// TIA Portal V19 export
// export: Created 2024-12-12T07:14:08.2418782Z, ExportSetting WithDefaults, DisplayName Totally Integrated Automation Portal, DisplayVersion V19 Update 1, DisplayName TIA Portal Openness, DisplayVersion V19 Update 1, DisplayName TIA Portal Version Control Interface, DisplayVersion V19, DisplayName SINAMICS Startdrive Advanced, DisplayVersion V19, DisplayName SINAMICS DCC, DisplayVersion V19, DisplayName SINAMICS Startdrive G130, G150, S120, S150, SINAMICS MV, G220, S200, S210, DisplayVersion V19, DisplayName SINAMICS Startdrive G110M, G120, G120C, G120D, G120P, G115D, DisplayVersion V19, DisplayName STEP 7 Professional, DisplayVersion V19 Update 1, DisplayName STEP 7 Safety, DisplayVersion V19 Update 1, DisplayName WinCC Advanced, DisplayVersion V19 Update 1, DisplayName WinCC Advanced / Unified PC, DisplayVersion V19 Update 1
DATA_BLOCK "DP1"   // DB30
{ S7_Optimized_Access := 'TRUE' }
VERSION : 0.1
// stored: AutoNumber true, DBAccessibleFromOPCUA true, DBAccessibleFromWebserver true, InstanceOfName DP_Exchange, InstanceOfType UDT, IsOnlyStoredInLoadMemory false, IsWriteProtectedInAS false
"DP_Exchange"
   // VAR RETAIN
   //    ExchangeToChain : "DP_Exchange_ToChain";
   //    ExchangeFromChain : "DP_Exchange_FromChain";
   //    Std : "DP_Exchange_Std";
   // END_VAR
BEGIN
   ExchangeToChain.Communication.RunMode := TRUE;
   ExchangeToChain.Communication.ConnectionFaulted := FALSE;
   ExchangeToChain.Work.Depositor := FALSE;
   ExchangeToChain.Work.TempDetect := FALSE;
   ExchangeToChain.Work.Vibrators := FALSE;
   ExchangeToChain.WorkedBy.Depositor := FALSE;
   ExchangeToChain.WorkedBy.TempDetect := FALSE;
   ExchangeToChain.WorkedBy.Vibrators := FALSE;
   ExchangeToChain.OutChainObstruction.Depositor := TRUE;
   ExchangeToChain.OutChainObstruction.TempDetect := TRUE;
   ExchangeToChain.OutChainObstruction.Vibrators := TRUE;
   ExchangeToChain.TimeWork.Depositor := 0;
   ExchangeToChain.TimeWork.Vibrator1 := 0;
   ExchangeToChain.TimeWork.Vibrator2 := 0;
   ExchangeToChain.TimeWork.VIbrator3 := 0;
   ExchangeToChain.AlmOKImmStopChain := TRUE;
   ExchangeToChain.Set_StrobeWorkReq := FALSE;
   ExchangeToChain.Set_StrobeWorkReqMouldBlock := FALSE;
   ExchangeToChain.RejByCycleInterruption := FALSE;
   ExchangeToChain.ChangeSpeedEna := TRUE;
   ExchangeToChain.MarkedByOpe := FALSE;
   ExchangeToChain.PresMould := FALSE;
   ExchangeToChain.Starved := FALSE;
   ExchangeToChain.DepositorEnabled := TRUE;
   ExchangeToChain.TempDetectorEnabled := TRUE;
   ExchangeToChain.LocalModeReq := FALSE;
   ExchangeToChain.Weight_StopInPhaseReq := TRUE;
   ExchangeToChain.Weight_AcusticReq := TRUE;
   ExchangeToChain.NoDoseAllowed := FALSE;
   ExchangeToChain."Dint"[0..4] := 0;
   ExchangeToChain.TempDetect_ScaledValue := 25.82104;
   ExchangeToChain.VMasterAtCycleEnd := 312.455;
   ExchangeToChain.VMasterRegPos := 0.0;
   ExchangeToChain.Infeed_VMasterRegPos1 := 0.0;
   ExchangeToChain.Infeed_VMasterRegPos2 := 0.0;
   ExchangeToChain.Outfeed_VMasterRegPos1 := 0.0;
   ExchangeToChain.Outfeed_VMasterRegPos2 := 0.0;
   ExchangeFromChain.Communication.RunMode := TRUE;
   ExchangeFromChain.Communication.ConnectionFaulted := FALSE;
   ExchangeFromChain.Chain.EnableMove := TRUE;
   ExchangeFromChain.Chain.StrobeWorkReq := FALSE;
   ExchangeFromChain.Chain.StrobeWorkReqMouldBlock := FALSE;
   ExchangeFromChain.Chain.CheckObstruction := FALSE;
   ExchangeFromChain.Chain.MoveInMan := FALSE;
   ExchangeFromChain.Chain.VMasterInPosition := TRUE;
   ExchangeFromChain.Chain.VMasterAtSpeed := FALSE;
   ExchangeFromChain.Chain.Cfg_1Jog_0Move := FALSE;
   ExchangeFromChain.ReqWork.Depositor := FALSE;
   ExchangeFromChain.ReqWork.TempDetect := FALSE;
   ExchangeFromChain.ReqWork.Vibrators := TRUE;
   ExchangeFromChain.SetWorkedBy.Depositor := FALSE;
   ExchangeFromChain.SetWorkedBy.TempDetect := FALSE;
   ExchangeFromChain.SetWorkedBy.Vibrators := FALSE;
   ExchangeFromChain.Set_MarkedByOpe := FALSE;
   ExchangeFromChain.Set_RejByCycleInterruption := FALSE;
   ExchangeFromChain.ChangeSpeedReq := FALSE;
   ExchangeFromChain.LocalModeActived := FALSE;
   ExchangeFromChain.LocalAbortReq := FALSE;
   ExchangeFromChain.Selected := TRUE;
   ExchangeFromChain."Dint"[0..4] := 0;
   ExchangeFromChain.SetPointSpeed := 25.0;
   ExchangeFromChain.ActualSpeed := 0.0;
   Std.ExchangeToGlobal.Communication.RunMode := TRUE;
   Std.ExchangeToGlobal.Communication.ConnectionFaulted := FALSE;
   Std.ExchangeToGlobal.Gen.Communication := FALSE;
   Std.ExchangeToGlobal.Gen.Selected := TRUE;
   Std.ExchangeToGlobal.Gen.Extracted := FALSE;
   Std.ExchangeToGlobal.Gen.EnaReq := FALSE;
   Std.ExchangeToGlobal.Gen.StaReq := FALSE;
   Std.ExchangeToGlobal.Gen.Started := FALSE;
   Std.ExchangeToGlobal.Gen.Unsuspended := FALSE;
   Std.ExchangeToGlobal.Gen.Ena_Suspended := TRUE;
   Std.ExchangeToGlobal.Gen.sts_Starting := FALSE;
   Std.ExchangeToGlobal.Gen.sts_Stopping := FALSE;
   Std.ExchangeToGlobal.Gen.sts_Aborting := FALSE;
   Std.ExchangeToGlobal.Gen.sts_Suspending := FALSE;
   Std.ExchangeToGlobal.Gen.sts_Unsuspending := FALSE;
   Std.ExchangeToGlobal.Gen.sts_Execute := FALSE;
   Std.ExchangeToGlobal.Gen.sts_Idle := TRUE;
   Std.ExchangeToGlobal.Gen.sts_Stopped := FALSE;
   Std.ExchangeToGlobal.Gen.sts_Aborted := FALSE;
   Std.ExchangeToGlobal.Gen.sts_Suspended := FALSE;
   Std.ExchangeToGlobal.Gen.sts_ModeManual := FALSE;
   Std.ExchangeToGlobal.Gen.sts_ModeAutomatic := TRUE;
   Std.ExchangeToGlobal.Gen.NewAlm := FALSE;
   Std.ExchangeToGlobal.Gen.NewSign := FALSE;
   Std.ExchangeToGlobal.Gen.RecipeOnlineLoadDone := FALSE;
   Std.ExchangeToGlobal.Gen.RecipeOnlineSaveDone := FALSE;
   Std.ExchangeToGlobal.Gen.RecipeOfflineLoadDone := FALSE;
   Std.ExchangeToGlobal.Gen.RecipeOfflineSaveDone := FALSE;
   Std.ExchangeToGlobal.Gen.LastHmiDataLoadDone := FALSE;
   Std.ExchangeToGlobal.Gen.LastHmiDataSaveDone := FALSE;
   Std.ExchangeToGlobal.Gen.InverterDiagnosticDone := FALSE;
   Std.ExchangeToGlobal.Gen.CmdMode := 1;
   Std.ExchangeToGlobal.Gen.Mode := 1;
   Std.ExchangeToGlobal.Gen.DisableEnaPbt := 0;
   Std.ExchangeToGlobal.Input.StaPbt := FALSE;
   Std.ExchangeToGlobal.Input.StoPbt := FALSE;
   Std.ExchangeToGlobal.Input.RstPbt := FALSE;
   Std.ExchangeToGlobal.Input.EnaPbt := FALSE;
   Std.ExchangeToGlobal.Input._4 := FALSE;
   Std.ExchangeToGlobal.Input._5 := FALSE;
   Std.ExchangeToGlobal.Input._6 := FALSE;
   Std.ExchangeToGlobal.Input._7 := FALSE;
   Std.ExchangeToGlobal.Input._8 := FALSE;
   Std.ExchangeToGlobal.Input._9 := FALSE;
   Std.ExchangeToGlobal.Input._10 := FALSE;
   Std.ExchangeToGlobal.Input._11 := FALSE;
   Std.ExchangeToGlobal.Input._12 := FALSE;
   Std.ExchangeToGlobal.Input._13 := FALSE;
   Std.ExchangeToGlobal.Input._14 := FALSE;
   Std.ExchangeToGlobal.Input._15 := FALSE;
   Std.ExchangeToGlobal.AlmOk.ThSwitch := TRUE;
   Std.ExchangeToGlobal.AlmOk.SafeComm := TRUE;
   Std.ExchangeToGlobal.AlmOk.SafeEmg := TRUE;
   Std.ExchangeToGlobal.AlmOk.SafeGuards := TRUE;
   Std.ExchangeToGlobal.AlmOk.GtaAirGroup := TRUE;
   Std.ExchangeToGlobal.AlmOk.Major := TRUE;
   Std.ExchangeToGlobal.AlmOk.Minor := TRUE;
   Std.ExchangeToGlobal.AlmOk.Spare07 := TRUE;
   Std.ExchangeToGlobal.AlmOk.Spare08 := TRUE;
   Std.ExchangeToGlobal.AlmOk.Spare09 := TRUE;
   Std.ExchangeToGlobal.AlmOk.Spare10 := TRUE;
   Std.ExchangeToGlobal.AlmOk.Spare11 := TRUE;
   Std.ExchangeToGlobal.AlmOk.Spare12 := TRUE;
   Std.ExchangeToGlobal.AlmOk.Spare13 := TRUE;
   Std.ExchangeToGlobal.AlmOk.Spare14 := TRUE;
   Std.ExchangeToGlobal.AlmOk.Spare15 := TRUE;
   Std.ExchangeToGlobal.AlmOk.Spare16 := TRUE;
   Std.ExchangeToGlobal.AlmOk.Spare17 := TRUE;
   Std.ExchangeToGlobal.AlmOk.Spare18 := TRUE;
   Std.ExchangeToGlobal.AlmOk.Spare19 := TRUE;
   Std.ExchangeToGlobal.AlmOk.Spare20 := TRUE;
   Std.ExchangeToGlobal.AlmOk.Spare21 := TRUE;
   Std.ExchangeToGlobal.AlmOk.Spare22 := TRUE;
   Std.ExchangeToGlobal.AlmOk.Spare23 := TRUE;
   Std.ExchangeToGlobal.AlmOk.Spare24 := TRUE;
   Std.ExchangeToGlobal.AlmOk.Spare25 := TRUE;
   Std.ExchangeToGlobal.AlmOk.Spare26 := TRUE;
   Std.ExchangeToGlobal.AlmOk.Spare27 := TRUE;
   Std.ExchangeToGlobal.AlmOk.Spare28 := TRUE;
   Std.ExchangeToGlobal.AlmOk.Spare29 := TRUE;
   Std.ExchangeToGlobal.AlmOk.Spare30 := TRUE;
   Std.ExchangeToGlobal.AlmOk.Spare31 := TRUE;
   Std.ExchangeToGlobal.AlmCauseOk.Ope := TRUE;
   Std.ExchangeToGlobal.AlmCauseOk.Ust := TRUE;
   Std.ExchangeToGlobal.AlmCauseOk.Dst := TRUE;
   Std.ExchangeToGlobal.AlmCauseOk.Ext := TRUE;
   Std.ExchangeToGlobal.AlmCauseOk.Mac := TRUE;
   Std.ExchangeToGlobal.AlmCauseOk.Spare05 := TRUE;
   Std.ExchangeToGlobal.AlmCauseOk.Spare06 := TRUE;
   Std.ExchangeToGlobal.AlmCauseOk.Spare07 := TRUE;
   Std.ExchangeToGlobal.AlmCauseOk.Spare08 := TRUE;
   Std.ExchangeToGlobal.AlmCauseOk.Spare09 := TRUE;
   Std.ExchangeToGlobal.AlmCauseOk.Spare10 := TRUE;
   Std.ExchangeToGlobal.AlmCauseOk.Spare11 := TRUE;
   Std.ExchangeToGlobal.AlmCauseOk.Spare12 := TRUE;
   Std.ExchangeToGlobal.AlmCauseOk.Spare13 := TRUE;
   Std.ExchangeToGlobal.AlmCauseOk.Spare14 := TRUE;
   Std.ExchangeToGlobal.AlmCauseOk.Spare15 := TRUE;
   Std.ExchangeToGlobal.AlmCauseOk.Spare16 := TRUE;
   Std.ExchangeToGlobal.AlmCauseOk.Spare17 := TRUE;
   Std.ExchangeToGlobal.AlmCauseOk.Spare18 := TRUE;
   Std.ExchangeToGlobal.AlmCauseOk.Spare19 := TRUE;
   Std.ExchangeToGlobal.AlmCauseOk.Spare20 := TRUE;
   Std.ExchangeToGlobal.AlmCauseOk.Spare21 := TRUE;
   Std.ExchangeToGlobal.AlmCauseOk.Spare22 := TRUE;
   Std.ExchangeToGlobal.AlmCauseOk.Spare23 := TRUE;
   Std.ExchangeToGlobal.AlmCauseOk.Spare24 := TRUE;
   Std.ExchangeToGlobal.AlmCauseOk.Spare25 := TRUE;
   Std.ExchangeToGlobal.AlmCauseOk.Spare26 := TRUE;
   Std.ExchangeToGlobal.AlmCauseOk.Spare27 := TRUE;
   Std.ExchangeToGlobal.AlmCauseOk.Spare28 := TRUE;
   Std.ExchangeToGlobal.AlmCauseOk.Spare29 := TRUE;
   Std.ExchangeToGlobal.AlmCauseOk.Spare30 := TRUE;
   Std.ExchangeToGlobal.AlmCauseOk.Spare31 := TRUE;
   Std.ExchangeToGlobal.AlmBannerFbk.FirstAlmDetection := FALSE;
   Std.ExchangeToGlobal.AlmBannerFbk.AlmPriority := 100;
   Std.ExchangeToGlobal.AlmBannerFbk.AlmCategory := -1;
   Std.ExchangeToGlobal.AlmBannerFbk.AlmCause := -1;
   Std.ExchangeToGlobal.AlmBannerFbk.AlmID := -1;
   Std.ExchangeToGlobal.AlmBannerFbk.GlobalAbsTime := 0;
   Std.ExchangeToGlobal.SignBannerFbk.SignPriority := 100;
   Std.ExchangeToGlobal.SignBannerFbk.SignCategory := -1;
   Std.ExchangeToGlobal.SignBannerFbk.SignID := -1;
   Std.ExchangeToGlobal.ExtCPU.PushButton.StaPbt := FALSE;
   Std.ExchangeToGlobal.ExtCPU.PushButton.StoPbt := FALSE;
   Std.ExchangeToGlobal.ExtCPU.PushButton.RstPbt := FALSE;
   Std.ExchangeToGlobal.ExtCPU.PushButton.EnaPbt := FALSE;
   Std.ExchangeToGlobal.ExtCPU.PushButton.EnaReq := FALSE;
   Std.ExchangeToGlobal.ExtCPU.PushButton.EnaStaReq := FALSE;
   Std.ExchangeToGlobal.ExtCPU.DeviceDiagDone := TRUE;
   Std.ExchangeToGlobal.ExtCPU.InverterDiagDone := FALSE;
   Std.ExchangeToGlobal.LightSiren.Cfg_StaPbt := 12515;
   Std.ExchangeToGlobal.LightSiren.Cfg_RstPbt := -1;
   Std.ExchangeToGlobal.LightSiren.Cfg_EnaPbt := 12515;
   Std.ExchangeToGlobal.LightSiren.Cfg_Siren := 3;
   Std.ExchangeToGlobal.LightSiren.Cfg_Stack := 3;
   Std.ExchangeToGlobal.LightSiren.Steady.StaPbtLgh := FALSE;
   Std.ExchangeToGlobal.LightSiren.Steady.RstPbtLgh := FALSE;
   Std.ExchangeToGlobal.LightSiren.Steady.EnaPbtLgh := FALSE;
   Std.ExchangeToGlobal.LightSiren.Steady.Siren := FALSE;
   Std.ExchangeToGlobal.LightSiren.Steady.YelStkLgh := FALSE;
   Std.ExchangeToGlobal.LightSiren.Steady.BluStkLgh := FALSE;
   Std.ExchangeToGlobal.LightSiren.Steady.GrnStkLgh := FALSE;
   Std.ExchangeToGlobal.LightSiren.Steady.WhtStkLgh := FALSE;
   Std.ExchangeToGlobal.LightSiren.Steady.Cust1_StaPbtLgh := FALSE;
   Std.ExchangeToGlobal.LightSiren.Steady.Cust1_RstPbtLgh := FALSE;
   Std.ExchangeToGlobal.LightSiren.Steady.Cust1_Siren := FALSE;
   Std.ExchangeToGlobal.LightSiren.Steady.Cust1_RedStkLgh := FALSE;
   Std.ExchangeToGlobal.LightSiren.Steady.Cust1_OngStkLgh := FALSE;
   Std.ExchangeToGlobal.LightSiren.Steady.Cust1_GrnStkLgh := FALSE;
   Std.ExchangeToGlobal.LightSiren.Steady.Cust1_BluStkLgh := FALSE;
   Std.ExchangeToGlobal.LightSiren.Steady.Cust1_WhtStkLgh := FALSE;
   Std.ExchangeToGlobal.LightSiren.Frequency1.StaPbtLgh := FALSE;
   Std.ExchangeToGlobal.LightSiren.Frequency1.RstPbtLgh := FALSE;
   Std.ExchangeToGlobal.LightSiren.Frequency1.EnaPbtLgh := FALSE;
   Std.ExchangeToGlobal.LightSiren.Frequency1.Siren := FALSE;
   Std.ExchangeToGlobal.LightSiren.Frequency1.YelStkLgh := FALSE;
   Std.ExchangeToGlobal.LightSiren.Frequency1.BluStkLgh := FALSE;
   Std.ExchangeToGlobal.LightSiren.Frequency1.GrnStkLgh := FALSE;
   Std.ExchangeToGlobal.LightSiren.Frequency1.WhtStkLgh := FALSE;
   Std.ExchangeToGlobal.LightSiren.Frequency1.Cust1_StaPbtLgh := FALSE;
   Std.ExchangeToGlobal.LightSiren.Frequency1.Cust1_RstPbtLgh := FALSE;
   Std.ExchangeToGlobal.LightSiren.Frequency1.Cust1_Siren := FALSE;
   Std.ExchangeToGlobal.LightSiren.Frequency1.Cust1_RedStkLgh := FALSE;
   Std.ExchangeToGlobal.LightSiren.Frequency1.Cust1_OngStkLgh := FALSE;
   Std.ExchangeToGlobal.LightSiren.Frequency1.Cust1_GrnStkLgh := FALSE;
   Std.ExchangeToGlobal.LightSiren.Frequency1.Cust1_BluStkLgh := FALSE;
   Std.ExchangeToGlobal.LightSiren.Frequency1.Cust1_WhtStkLgh := FALSE;
   Std.ExchangeToGlobal.LightSiren.Frequency2.StaPbtLgh := FALSE;
   Std.ExchangeToGlobal.LightSiren.Frequency2.RstPbtLgh := FALSE;
   Std.ExchangeToGlobal.LightSiren.Frequency2.EnaPbtLgh := FALSE;
   Std.ExchangeToGlobal.LightSiren.Frequency2.Siren := FALSE;
   Std.ExchangeToGlobal.LightSiren.Frequency2.YelStkLgh := FALSE;
   Std.ExchangeToGlobal.LightSiren.Frequency2.BluStkLgh := FALSE;
   Std.ExchangeToGlobal.LightSiren.Frequency2.GrnStkLgh := FALSE;
   Std.ExchangeToGlobal.LightSiren.Frequency2.WhtStkLgh := FALSE;
   Std.ExchangeToGlobal.LightSiren.Frequency2.Cust1_StaPbtLgh := FALSE;
   Std.ExchangeToGlobal.LightSiren.Frequency2.Cust1_RstPbtLgh := FALSE;
   Std.ExchangeToGlobal.LightSiren.Frequency2.Cust1_Siren := FALSE;
   Std.ExchangeToGlobal.LightSiren.Frequency2.Cust1_RedStkLgh := FALSE;
   Std.ExchangeToGlobal.LightSiren.Frequency2.Cust1_OngStkLgh := FALSE;
   Std.ExchangeToGlobal.LightSiren.Frequency2.Cust1_GrnStkLgh := FALSE;
   Std.ExchangeToGlobal.LightSiren.Frequency2.Cust1_BluStkLgh := FALSE;
   Std.ExchangeToGlobal.LightSiren.Frequency2.Cust1_WhtStkLgh := FALSE;
   Std.ExchangeToGlobal.LightSiren.Frequency3.StaPbtLgh := FALSE;
   Std.ExchangeToGlobal.LightSiren.Frequency3.RstPbtLgh := FALSE;
   Std.ExchangeToGlobal.LightSiren.Frequency3.EnaPbtLgh := FALSE;
   Std.ExchangeToGlobal.LightSiren.Frequency3.Siren := FALSE;
   Std.ExchangeToGlobal.LightSiren.Frequency3.YelStkLgh := FALSE;
   Std.ExchangeToGlobal.LightSiren.Frequency3.BluStkLgh := FALSE;
   Std.ExchangeToGlobal.LightSiren.Frequency3.GrnStkLgh := FALSE;
   Std.ExchangeToGlobal.LightSiren.Frequency3.WhtStkLgh := FALSE;
   Std.ExchangeToGlobal.LightSiren.Frequency3.Cust1_StaPbtLgh := FALSE;
   Std.ExchangeToGlobal.LightSiren.Frequency3.Cust1_RstPbtLgh := FALSE;
   Std.ExchangeToGlobal.LightSiren.Frequency3.Cust1_Siren := FALSE;
   Std.ExchangeToGlobal.LightSiren.Frequency3.Cust1_RedStkLgh := FALSE;
   Std.ExchangeToGlobal.LightSiren.Frequency3.Cust1_OngStkLgh := FALSE;
   Std.ExchangeToGlobal.LightSiren.Frequency3.Cust1_GrnStkLgh := FALSE;
   Std.ExchangeToGlobal.LightSiren.Frequency3.Cust1_BluStkLgh := FALSE;
   Std.ExchangeToGlobal.LightSiren.Frequency3.Cust1_WhtStkLgh := FALSE;
   Std.ExchangeToGlobal.LightSiren.Frequency4.StaPbtLgh := FALSE;
   Std.ExchangeToGlobal.LightSiren.Frequency4.RstPbtLgh := FALSE;
   Std.ExchangeToGlobal.LightSiren.Frequency4.EnaPbtLgh := FALSE;
   Std.ExchangeToGlobal.LightSiren.Frequency4.Siren := FALSE;
   Std.ExchangeToGlobal.LightSiren.Frequency4.YelStkLgh := FALSE;
   Std.ExchangeToGlobal.LightSiren.Frequency4.BluStkLgh := FALSE;
   Std.ExchangeToGlobal.LightSiren.Frequency4.GrnStkLgh := FALSE;
   Std.ExchangeToGlobal.LightSiren.Frequency4.WhtStkLgh := FALSE;
   Std.ExchangeToGlobal.LightSiren.Frequency4.Cust1_StaPbtLgh := FALSE;
   Std.ExchangeToGlobal.LightSiren.Frequency4.Cust1_RstPbtLgh := FALSE;
   Std.ExchangeToGlobal.LightSiren.Frequency4.Cust1_Siren := FALSE;
   Std.ExchangeToGlobal.LightSiren.Frequency4.Cust1_RedStkLgh := FALSE;
   Std.ExchangeToGlobal.LightSiren.Frequency4.Cust1_OngStkLgh := FALSE;
   Std.ExchangeToGlobal.LightSiren.Frequency4.Cust1_GrnStkLgh := FALSE;
   Std.ExchangeToGlobal.LightSiren.Frequency4.Cust1_BluStkLgh := FALSE;
   Std.ExchangeToGlobal.LightSiren.Frequency4.Cust1_WhtStkLgh := FALSE;
   Std.ExchangeToGlobal.PackML.Sts_Aborted := FALSE;
   Std.ExchangeToGlobal.PackML.Sts_Aborting := FALSE;
   Std.ExchangeToGlobal.PackML.Sts_Clearing := FALSE;
   Std.ExchangeToGlobal.PackML.Sts_Complete := FALSE;
   Std.ExchangeToGlobal.PackML.Sts_Completing := FALSE;
   Std.ExchangeToGlobal.PackML.Sts_Execute := FALSE;
   Std.ExchangeToGlobal.PackML.Sts_Held := FALSE;
   Std.ExchangeToGlobal.PackML.Sts_Holding := FALSE;
   Std.ExchangeToGlobal.PackML.Sts_Idle := TRUE;
   Std.ExchangeToGlobal.PackML.Sts_Resetting := FALSE;
   Std.ExchangeToGlobal.PackML.Sts_Starting := FALSE;
   Std.ExchangeToGlobal.PackML.Sts_Stopped := FALSE;
   Std.ExchangeToGlobal.PackML.Sts_Stopping := FALSE;
   Std.ExchangeToGlobal.PackML.Sts_Suspended := FALSE;
   Std.ExchangeToGlobal.PackML.Sts_Suspending := FALSE;
   Std.ExchangeToGlobal.PackML.Sts_UnHolding := FALSE;
   Std.ExchangeToGlobal.PackML.Sts_UnSuspending := FALSE;
   Std.ExchangeToGlobal.PackML.Sts_AbortedEnabled := TRUE;
   Std.ExchangeToGlobal.PackML.Sts_AbortingEnabled := TRUE;
   Std.ExchangeToGlobal.PackML.Sts_ClearingEnabled := TRUE;
   Std.ExchangeToGlobal.PackML.Sts_CompleteEnabled := FALSE;
   Std.ExchangeToGlobal.PackML.Sts_CompletingEnabled := FALSE;
   Std.ExchangeToGlobal.PackML.Sts_ExecuteEnabled := TRUE;
   Std.ExchangeToGlobal.PackML.Sts_HeldEnabled := FALSE;
   Std.ExchangeToGlobal.PackML.Sts_HoldingEnabled := FALSE;
   Std.ExchangeToGlobal.PackML.Sts_IdleEnabled := TRUE;
   Std.ExchangeToGlobal.PackML.Sts_ResettingEnabled := TRUE;
   Std.ExchangeToGlobal.PackML.Sts_StartingEnabled := TRUE;
   Std.ExchangeToGlobal.PackML.Sts_StoppedEnabled := TRUE;
   Std.ExchangeToGlobal.PackML.Sts_StoppingEnabled := TRUE;
   Std.ExchangeToGlobal.PackML.Sts_SuspendedEnabled := TRUE;
   Std.ExchangeToGlobal.PackML.Sts_SuspendingEnabled := TRUE;
   Std.ExchangeToGlobal.PackML.Sts_UnHoldingEnabled := FALSE;
   Std.ExchangeToGlobal.PackML.Sts_UnSuspendingEnabled := TRUE;
   Std.ExchangeToGlobal.SignOk := TRUE;
   Std.ExchangeToGlobal."Dint"[0..4] := 0;
END_DATA_BLOCK
